FUNCTION_BLOCK Delta
VAR_INPUT
	MotionParameters	: DeltaMotionParameters_typ;			// Motion parameters used by internal motion function blocks	
	myMCSOverride: LREAL := 10.0;
	xSetOverride: BOOL;
	lrGrpOverride: MC_LREAL := 1.0;
	fbMC_GroupSetOverride : MC_GroupSetOverride;		
END_VAR

VAR_OUTPUT
	
	Ready				: BOOL;
	Busy				: BOOL;
	
	Error				: BOOL;
	ErrorID				: UDINT;
	ErrorOrigin			: STRING;	
		
	internalKinChanNCtoPLC	AT %I* : NCTOPLC_NCICHANNEL_REF;
	internalKinChanPLCtoNC	AT %Q* : PLCTONC_NCICHANNEL_REF;
		btest2: BOOL;	
	InKinematicsGroup		: BOOL;	
	InCoordinatedGroup		: BOOL;
	
	InSyncWithConveyor		: BOOL;

	//IdentInKinGroup			: UDINT;
	//IdentInCMGroup			: UDINT; 	
	
	ACS_A_REF	: AXIS_REF;
	ACS_B_REF	: AXIS_REF;
	ACS_C_REF	: AXIS_REF;
	
	MCS_X_REF	: AXIS_REF;
	MCS_Y_REF	: AXIS_REF;
	MCS_Z_REF	: AXIS_REF;
END_VAR
VAR
	
	{attribute 'instance-path'}
	{attribute 'no-init'}
	InstancePath			: STRING;
	btest: BOOL;
	AirVariable				AT %Q* : BOOL;
	
	internalEnable			: BOOL;
	internalDisable			: BOOL;
	
	//internalCurrentMoveType	: DeltaCommandType_enum;
	
	internalState			: DeltaState_enum;
	
	internalSetCoordTrafoDone	: BOOL;
	internalMovePathDone		: BOOL;

	
	internalInitObjPos		: ARRAY [1..3] OF MC_LREAL := [0,0,0];
	internalAxesList		: ST_KinAxes;
	internalCMGroup			: AXES_GROUP_REF;
	
	internalTrackAxis		: REFERENCE TO AXIS_REF;
	
	internalPathBuffer		: ARRAY[0..32767] OF BYTE;
	internalPathData		: MC_PATH_DATA_REF( ADR( internalPathBuffer ), SIZEOF( internalPathBuffer ));
		
	externalRoute			: REFERENCE TO Route;	

	internalActiveCoordRef	: MC_COORD_REF;		

	// Internal function blocks
	fbReset_MCS_X			: MC_Reset;
	fbReset_MCS_Y			: MC_Reset;
	fbReset_MCS_Z			: MC_Reset;
	
	fbReset_ACS_A			: MC_Reset;
	fbReset_ACS_B			: MC_Reset;
	fbReset_ACS_C			: MC_Reset;
	
	fbPower_MCS_X			: MC_Power;
	fbPower_MCS_Y			: MC_Power;
	fbPower_MCS_Z			: MC_Power;
	
	fbPower_ACS_A			: MC_Power;
	fbPower_ACS_B			: MC_Power;
	fbPower_ACS_C			: MC_Power;	
	
	fbAddAxisToGrp			: ARRAY[0..2] OF MC_AddAxisToGroup;
	fbGroupEnable			: MC_GroupEnable;
	
	fbKinConfigGroup		: FB_KinConfigGroup; 
	fbKinResetGroup			: FB_KinResetGroup;
	
	fbTrackBelt				: MC_TrackConveyorBelt;
	
	fbSetCoordTrafo			: MC_SetCoordinateTransform;
	fbMoveLinearPrep		: MC_MoveLinearAbsolutePreparation;
	fbMovePath				: MC_MovePath;
	fbMovePathExt			: MC_MovePath;
END_VAR

METHOD Cyclic : BOOL
VAR_IN_OUT
	//	KinematicGroup		: NCTOPLC;
END_VAR
VAR
	i: USINT;

END_VAR
CASE internalState OF
	DL_IDLE:	// ------------------------------------------------------- idle state
	
		Ready		:= FALSE;
		Busy		:= FALSE;
		
		internalDisable		:= FALSE;
		IF internalEnable THEN
			internalEnable		:= FALSE;
			internalState		:= DL_RESET;
		END_IF
	
	DL_RESET:	// ------------------------------------------------------- resets all axis objects
	
		Ready		:= FALSE;
		Busy		:= TRUE;
		Error		:= FALSE;
		ErrorID		:= 0;
		
		fbReset_MCS_X.Execute		:= TRUE;
		fbReset_MCS_Y.Execute		:= TRUE;
		fbReset_MCS_Z.Execute		:= TRUE;		
		
		fbReset_ACS_A.Execute		:= TRUE;
		fbReset_ACS_B.Execute		:= TRUE;
		fbReset_ACS_C.Execute		:= TRUE;
		
		IF fbReset_MCS_X.Done AND
			fbReset_MCS_Y.Done AND
			fbReset_MCS_Z.Done AND
			fbReset_ACS_A.Done AND
			fbReset_ACS_B.Done AND
			fbReset_ACS_C.Done THEN
			
			fbReset_MCS_X.Execute		:= FALSE;
			fbReset_MCS_Y.Execute		:= FALSE;
			fbReset_MCS_Z.Execute		:= FALSE;		
		
			fbReset_ACS_A.Execute		:= FALSE;
			fbReset_ACS_B.Execute		:= FALSE;
			fbReset_ACS_C.Execute		:= FALSE;
			
			internalState	:= DL_POWER_AXES;
			
		ELSIF fbReset_MCS_X.Error OR
			fbReset_MCS_Y.Error OR
			fbReset_MCS_Z.Error OR
			fbReset_ACS_A.Error OR
			fbReset_ACS_B.Error OR
			fbReset_ACS_C.Error THEN
			
			ErrorID; // TODO add whatever the error was for that block
			ErrorOrigin		:= CONCAT( InstancePath, '.fbReset' );
			internalState	:= DL_ERROR; 		
		END_IF
		
	DL_POWER_AXES:	// --------------------------------------------------- energizes all axis objects
	
		Ready		:= FALSE;
		Busy		:= TRUE;
		Error		:= FALSE;
		ErrorID		:= 0;

			fbPower_MCS_X.Enable	:= TRUE;
			fbPower_MCS_Y.Enable	:= TRUE;
			fbPower_MCS_Z.Enable	:= TRUE;
			
			fbPower_MCS_X.Enable_Positive	:= TRUE;
			fbPower_MCS_Y.Enable_Positive	:= TRUE;
			fbPower_MCS_Z.Enable_Positive	:= TRUE;
			
			fbPower_MCS_X.Enable_Negative	:= TRUE;
			fbPower_MCS_Y.Enable_Negative	:= TRUE;
			fbPower_MCS_Z.Enable_Negative	:= TRUE;
			
			fbPower_ACS_A.Enable	:= TRUE;
			fbPower_ACS_B.Enable	:= TRUE;
			fbPower_ACS_C.Enable	:= TRUE;
			
			fbPower_ACS_A.Enable_Positive	:= TRUE;
			fbPower_ACS_B.Enable_Positive	:= TRUE;
			fbPower_ACS_C.Enable_Positive	:= TRUE;
			
			fbPower_ACS_A.Enable_Negative	:= TRUE;
			fbPower_ACS_B.Enable_Negative	:= TRUE;
			fbPower_ACS_C.Enable_Negative	:= TRUE;
			
			fbPower_MCS_X.Override		:= myMCSOverride;
			fbPower_MCS_Y.Override		:= myMCSOverride;
			fbPower_MCS_Z.Override		:= myMCSOverride;
			
			IF fbPower_MCS_X.Status AND
				fbPower_MCS_Y.Status AND
				fbPower_MCS_Z.Status AND
				fbPower_ACS_A.Status AND
				fbPower_ACS_B.Status AND
				fbPower_ACS_C.Status THEN
				
				internalState	:= DL_SET_IK;
				
			ELSIF fbPower_MCS_X.Error OR
				fbPower_MCS_Y.Error OR
				fbPower_MCS_Z.Error OR
				fbPower_ACS_A.Error OR
				fbPower_ACS_B.Error OR
				fbPower_ACS_C.Error THEN
				
				ErrorID;	// TODO add whatever the error was that block
				ErrorOrigin		:= CONCAT( InstancePath, '.fbPower');
				internalState	:= DL_ERROR;
			END_IF

	
	DL_SET_IK:	// ------------------------------------------------------- enables the inverse kinematics transformation
	
		Ready		:= FALSE;
		Busy		:= TRUE;
		Error		:= FALSE;
		ErrorID		:= 0;

		internalAxesList.nAxisIdsAcs[1]		:= ACS_A_REF.NcToPlc.AxisId;
		internalAxesList.nAxisIdsAcs[2]		:= ACS_B_REF.NcToPlc.AxisId;
		internalAxesList.nAxisIdsAcs[3]		:= ACS_C_REF.NcToPlc.AxisId;
		
		internalAxesList.nAxisIdsMcs[1]		:= MCS_X_REF.NcToPlc.AxisId;
		internalAxesList.nAxisIdsMcs[2]		:= MCS_Y_REF.NcToPlc.AxisId;
		internalAxesList.nAxisIdsMcs[3]		:= MCS_Z_REF.NcToPlc.AxisId;
		
		fbKinConfigGroup.bExecute			:= TRUE;
		fbKinConfigGroup.bCartesianMode		:= TRUE;
	
	
		IF fbKinConfigGroup.bDone THEN
		//	fbKinConfigGroup.bExecute		:= FALSE;
			internalState					:= DL_DEBUG; //DL_ADD_AXES_TO_CM; // 
		ELSIF fbKinConfigGroup.bError THEN
			ErrorID			:= fbKinConfigGroup.nErrorId;
			ErrorOrigin		:= CONCAT(InstancePath,'.fbKinConfigGroup');
			internalState	:= DL_ERROR;
		END_IF;

		
	DL_ADD_AXES_TO_CM:	// ----------------------------------------------- adds MCS axes to CM Group
	
		Ready		:= FALSE;
		Busy		:= TRUE;
		Error		:= FALSE;
		ErrorID		:= 0;

			fbAddAxisToGrp[0].IdentInGroup	:= MCS_X;
			// fbAddAxisToGrp[0].Axis			:= MCS_X_REF;
			
			fbAddAxisToGrp[1].IdentInGroup	:= MCS_Y;
			// fbAddAxisToGrp[1].Axis			:= MCS_Y_REF;	
			
			fbAddAxisToGrp[2].IdentInGroup	:= MCS_Z;
			// fbAddAxisToGrp[2].Axis			:= MCS_Z_REF;
			
			FOR i := 0 TO 2 DO
				fbAddAxisToGrp[i].Execute		:= TRUE;
			END_FOR
			
			IF fbAddAxisToGrp[0].Done AND
				fbAddAxisToGrp[1].Done AND
				fbAddAxisToGrp[2].Done THEN
				
				fbAddAxisToGrp[0].Execute	:= FALSE;
				fbAddAxisToGrp[1].Execute	:= FALSE;
				fbAddAxisToGrp[2].Execute	:= FALSE;
				
				internalState	:= DL_ENABLE_CM;
				
			ELSIF fbAddAxisToGrp[0].Error OR
				fbAddAxisToGrp[1].Error OR
				fbAddAxisToGrp[2].Error THEN
				
				fbAddAxisToGrp[0].Execute	:= FALSE;
				fbAddAxisToGrp[1].Execute	:= FALSE;
				fbAddAxisToGrp[2].Execute	:= FALSE;
				
				ErrorID;		// todo : add whichever block errored
				ErrorOrigin		:= CONCAT(InstancePath,'.fbAddAxisToGrp');
				internalState	:= DL_ERROR;
			END_IF

	DL_ENABLE_CM:	// ------------------------------------------------------- enables the coordinated motion group
	
		Ready		:= FALSE;
		Busy		:= TRUE;
		Error		:= FALSE;
		ErrorID		:= 0;
		
			fbGroupEnable.Execute		:= TRUE;
			
			IF fbGroupEnable.Done THEN
				internalState	:= DL_RUN;
			ELSIF fbGroupEnable.Error THEN
				ErrorID			:= fbGroupEnable.ErrorId;
				ErrorOrigin		:= CONCAT(InstancePath,'.fbGroupEnable');
				internalState	:= DL_ERROR;
			END_IF
		
	DL_RUN:	// --------------------------------------------------------------- Delta running, ready for commands
	
		Ready		:= TRUE;
		Busy		:= FALSE;
		Error		:= FALSE;
		ErrorID		:= 0;
				
		// reset all commanded function blocks when the execute is recieved
		IF fbSetCoordTrafo.Busy OR fbSetCoordtrafo.CommandAborted THEN
			fbSetCoordTrafo.Execute		:= FALSE;
		ELSIF fbMovePath.Busy OR fbMovePath.CommandAborted THEN
			fbMovePath.Execute			:= FALSE;
		ELSIF fbMovePathEXT.Busy OR fbMovePathEXT.CommandAborted THEN
			fbMovePath.Execute			:= FALSE;
		ELSIF fbTrackBelt.Active OR fbTrackBelt.CommandAborted THEN
			fbTrackBelt.Execute			:= FALSE;
		END_IF
		
		// and catch all internal function block errors
		IF fbSetCoordTrafo.Error THEN
			ErrorID			:= fbSetCoordTrafo.ErrorId;
			ErrorOrigin		:= CONCAT( InstancePath, '.fbSetCoordTrafo' );
			internalState	:= DL_ERROR;
		ELSIF fbMovePath.Error THEN
			ErrorID			:= fbMovePath.ErrorId;
			ErrorOrigin		:= CONCAT( InstancePath, '.fbMovePath' );
			internalState	:= DL_ERROR;
		ELSIF fbMovePathEXT.Error THEN
			ErrorID			:= fbMovePathEXT.ErrorId;
			ErrorOrigin		:= CONCAT( InstancePath, '.fbMovePathEXT' );
			internalState	:= DL_ERROR;
		ELSIF fbTrackBelt.Error THEN
			ErrorID			:= fbMovePath.ErrorId;
			ErrorOrigin		:= CONCAT( InstancePath, '.fbMovePath' );
			internalState	:= DL_ERROR;
		END_IF
	
	DL_ERROR:	// ----------------------------------------------------------- Error state
	
		Ready		:= FALSE;
		Busy		:= FALSE;
		Error		:= TRUE;
	
END_CASE

fbReset_ACS_A( Axis := ACS_A_REF );
fbReset_ACS_B( Axis := ACS_B_REF );
fbReset_ACS_C( Axis := ACS_C_REF );
fbReset_MCS_X( Axis := MCS_X_REF );
fbReset_MCS_Y( Axis := MCS_Y_REF );
fbReset_MCS_Z( Axis := MCS_Z_REF );

fbPower_ACS_A( Axis := ACS_A_REF );
fbPower_ACS_B( Axis := ACS_B_REF );
fbPower_ACS_C( Axis := ACS_C_REF );
fbPower_MCS_X( Axis := MCS_X_REF );
fbPower_MCS_Y( Axis := MCS_Y_REF );
fbPower_MCS_Z( Axis := MCS_Z_REF );

fbAddAxisToGrp[0]( AxesGroup := internalCMGroup, Axis := MCS_X_REF );
fbAddAxisToGrp[1]( AxesGroup := internalCMGroup, Axis := MCS_Y_REF );
fbAddAxisToGrp[2]( AxesGroup := internalCMGroup, Axis := MCS_Z_REF );

fbGroupEnable( AxesGroup := internalCMGroup );

fbKinConfigGroup( stAxesList := internalAxesList, stKinRefIn := internalKinChanNCtoPLC );
fbKinResetGroup( stKinRefIn := internalKinChanNCtoPLC, stAxesList := internalAxesList );

fbSetCoordTrafo( AxesGroup := internalCMGroup );

fbMovePath( AxesGroup := internalCMGroup, PathData := internalPathData );
fbMovePathEXT( AxesGroup := internalCMGroup, PathData := externalRoute.PathData );

fbMC_GroupSetOverride(
	AxesGroup:= internalCMGroup, 
	Enable:= xSetOverride, 
	VelFactor:= lrGrpOverride, 
	Enabled=> , 
	Busy=> , 
	Error=> , 
	ErrorId=> , 
	ActualVelFactor=> );
END_METHOD

METHOD Disable : BOOL
VAR_INPUT
END_VAR
END_METHOD

METHOD DisableAir : BOOL
VAR_INPUT
END_VAR
AirVariable	:= FALSE;
END_METHOD

METHOD Enable : BOOL
VAR_INPUT
END_VAR
IF internalState = DL_IDLE THEN
	internalEnable		:= TRUE;
END_IF;
END_METHOD

METHOD EnableAir : BOOL
VAR_INPUT
END_VAR
AirVariable	:= TRUE;
END_METHOD

METHOD ExecuteRoute : BOOL
VAR_INPUT
	Route		: REFERENCE TO Route;
END_VAR
externalRoute			REF= Route;
fbMovePathEXT.Execute	:= TRUE;
END_METHOD

METHOD MoveDirectTo : BOOL
VAR_INPUT
	X			: LREAL;
	Y			: LREAL;
	Z			: LREAL;
END_VAR
VAR
	posVector			: ARRAY[0..2] OF LREAL;
	toleranceBall		: ARRAY[0..1] OF LREAL;
END_VAR
// clear any existing waypoints in the path buffer
internalPathData.ClearPath();

// add a single point at the destination
posVector[0]	:= X;
posVector[1]	:= Y;
posVector[2]	:= Z;

// blending radii follows a ratio recommendation from infosys
toleranceBall[0]	:= 0.5 * MotionParameters.BlendingRadius;
toleranceBall[1]	:= MotionParameters.BlendingRadius;

fbMoveLinearPrep.Position			:= ADR( posVector );
fbMoveLinearPrep.PositionCount		:= 3;
fbMoveLinearPrep.Velocity			:= MotionParameters.Velocity;
fbMoveLinearPrep.Acceleration		:= MotionParameters.Acceleration;
fbMoveLinearPrep.Deceleration		:= MotionParameters.Deceleration;
fbMoveLinearPrep.Jerk				:= MotionParameters.Jerk;
fbMoveLinearPrep.BufferMode			:= mcBlendingPrevious;

fbMoveLinearPrep.TransitionMode				:= mcTransModeCornerDistanceAdvanced;
fbMoveLinearPrep.TransitionParameter		:= ADR( toleranceBall );
fbMoveLinearPrep.TransitionParameterCount	:= 2;
fbMoveLinearPrep.InvokeId					:= 100;

fbMoveLinearPrep( PathData := internalPathData );

// execute mc_movepath
fbMovePath.Execute	:= TRUE;

fbMovePath( AxesGroup := internalCMGroup, PathData := internalPathData );
END_METHOD

PROPERTY MovePathDone : BOOL
GET
MovePathDone		:= fbMovePath.Done;
END_GET
END_PROPERTY

METHOD Reset : BOOL
VAR_INPUT
END_VAR
internalState := DL_IDLE;
END_METHOD

METHOD ReturnHome : BOOL
VAR_INPUT
END_VAR
// Zero is home, right?
THIS^.MoveDirectTo( 0, 100, 50);
END_METHOD

METHOD SetAcceleration : BOOL
VAR_INPUT
	Acceleration	: LREAL;
END_VAR
// prevents a negative value from being accepted
MotionParameters.Acceleration		:= LIMIT( 0, Acceleration, 1E300 );
END_METHOD

METHOD SetCoordTrafo : BOOL
VAR_INPUT
	CoordRef	: MC_COORD_REF;
END_VAR
// Set the function block to change coordinate reference frame
fbSetCoordTrafo.Execute				:= TRUE;
fbSetCoordTrafo.CoordTransform		:= CoordRef;	

internalActiveCoordRef				:= CoordRef;

fbSetCoordTrafo( AxesGroup := internalCMGroup );
END_METHOD

PROPERTY SetCoordTrafoDone : BOOL
GET
SetCoordTrafoDone	:= fbSetCoordTrafo.Done;
END_GET
END_PROPERTY

METHOD SetDeceleration : BOOL
VAR_INPUT
	Deceleration		: LREAL;
END_VAR

// prevent a negative value from being accepted
MotionParameters.Deceleration	:= LIMIT( 0, Deceleration, 1E300 );
END_METHOD

METHOD SetJerk : BOOL
VAR_INPUT
	Jerk		: LREAL;
END_VAR

// Prevents a negative value from being accepted.
MotionParameters.Jerk		:= LIMIT( 0, Jerk, 1E300 );
END_METHOD

METHOD SetVelocity : BOOL
VAR_INPUT
	Velocity		: LREAL;
END_VAR

// Prevents a negative value from being accepted
MotionParameters.Velocity		:= LIMIT( 0, Velocity, 1E300 );
END_METHOD

METHOD TrackConveyor : BOOL
VAR_INPUT
	MasterRefPos		: MC_LREAL;
	TrackAxis			: REFERENCE TO AXIS_REF;
	CoordFrame			: MC_COORD_REF;
END_VAR


internalTrackAxis		REF= TrackAxis;

//initialObjectPos[1]		:= 0;
//initialObjectPos[2]		:= 0;
//initialObjectPos[3]		:= 0;

fbTrackBelt.CoordTransform			:= CoordFrame;
fbTrackBelt.InitialObjectPos		:= ADR( internalInitObjPos );
fbTrackBelt.InitialObjectPosCount	:= 3;
fbTrackBelt.MasterRefPos			:= MasterRefPos;

fbTrackBelt.Velocity		:= MotionParameters.Velocity;
fbTrackBelt.Acceleration	:= MotionParameters.Acceleration;
fbTrackBelt.Deceleration	:= MotionParameters.Deceleration;
fbTrackBelt.Jerk			:= MotionParameters.Jerk;

fbTrackBelt.Execute		:= TRUE;

fbTrackBelt( AxesGroup := internalCMGroup, ConveyorBelt := internalTrackAxis );
END_METHOD

PROPERTY TrackConveyorActive : BOOL
GET
TrackConveyorActive		:= fbTrackBelt.InSync;
END_GET
END_PROPERTY

METHOD TraverseAtHeightTo : BOOL
VAR_INPUT
	X			: LREAL;
	Y			: LREAL;
	Z			: LREAL;
	TraverseZ	: LREAL;
END_VAR
VAR
	posVector		: ARRAY[0..2] OF LREAL;
	toleranceBall	: ARRAY[0..1] OF LREAL;
END_VAR
// clear any existing waypoints in the path buffer
internalPathData.ClearPath();

toleranceBall[0]	:= 0.5 * MotionParameters.BlendingRadius;
toleranceBall[1]	:= MotionParameters.BlendingRadius;

fbMoveLinearPrep.PositionCount		:= 3;
fbMoveLinearPrep.Velocity			:= MotionParameters.Velocity;
fbMoveLinearPrep.Acceleration		:= MotionParameters.Acceleration;
fbMoveLinearPrep.Deceleration		:= MotionParameters.Deceleration;
fbMoveLinearPrep.Jerk				:= MotionParameters.Jerk;
fbMoveLinearPrep.BufferMode			:= mcBlendingPrevious;

fbMoveLinearPrep.TransitionMode				:= mcTransModeCornerDistanceAdvanced;
fbMoveLinearPrep.TransitionParameter		:= ADR( toleranceBall );
fbMoveLinearPrep.TransitionParameterCount	:= 2;
fbMoveLinearPrep.InvokeId					:= 100;

// add a vertical movement to the traverse height
posVector[0]		:= MCS_X_REF.NcToPlc.ActPos; 
posVector[1]		:= MCS_Y_REF.NcToPlc.ActPos;
posVector[2]		:= TraverseZ;

fbMoveLinearPrep.Position		:= ADR( posVector );
fbMoveLinearPrep( PathData := internalPathData );

// add a traversal move to a point above/below the destination
posVector[0]		:= X;	// destination X
posVector[1]		:= Y;	// destination Y
posVector[2]		:= TraverseZ;	// traversal height

fbMoveLinearPrep.Position		:= ADR( posVector );
fbMoveLinearPrep( PathData := internalPathData );

// add a vertical move to the destination itself
posVector[0]		:= X;
posVector[1]		:= Y;
posVector[2]		:= Z;

fbMoveLinearPrep.Position		:= ADR( posVector );
fbMoveLinearPrep( PathData := internalPathData );

// execute mc_movepath
fbMovePath.Execute	:= TRUE;

// Call once for Busy output
fbMovePath( AxesGroup := internalCMGroup, PathData := internalPathData );
END_METHOD

END_FUNCTION_BLOCK

(* stored: Version 1.1.0.1, ProductVersion 3.1.4024.11
   POU Delta: Id {492a738f-fc6d-4715-b733-4ea1b08e2312}, SpecialFunc None
   Folder Methods: Id {a2d46a1e-7a9e-44a1-9a9c-487d94df0d8d}
   Folder Properties: Id {68d119c4-1e71-4d9e-a63e-63c332a25cde}
   Method Cyclic: Id {08a56dcb-206a-41ec-ac0a-83b543ba62a8}
   Method Disable: Id {f8852278-a902-41fb-8b1a-a53ea61cbd64}
   Method DisableAir: Id {74258680-12ce-4520-8174-1e7920fb856e}
   Method Enable: Id {f4887e95-9084-4d7c-8994-4709154d6c02}
   Method EnableAir: Id {64a72ef1-4b6d-4e9c-8d63-cad412c5e0f0}
   Method ExecuteRoute: Id {0f1c4d90-fa0e-4ee0-9899-a01e330415e2}
   Method MoveDirectTo: Id {610f0aa4-e8d8-4a0e-b42c-d66003cd2595}
   Property MovePathDone: Id {dd8dbeba-3161-4047-8127-ea64b21675c1}
   Get Get: Id {7df17e80-557a-41df-8651-9ebd7ef9a364}
   Method Reset: Id {53b97b6c-d929-489a-b91b-ad9f50847a2c}
   Method ReturnHome: Id {4a762706-93bb-4e83-8b35-d2c1fae7dbb3}
   Method SetAcceleration: Id {92321fb0-df12-41a8-a2c8-436a5c15bd2a}
   Method SetCoordTrafo: Id {6bf0c707-36e2-400d-ba6a-1409a4ef623e}
   Property SetCoordTrafoDone: Id {71fa1ee3-447a-48eb-933c-e282e4815b89}
   Get Get: Id {dca464b8-bfd9-4ed6-aeb3-8b7143978587}
   Method SetDeceleration: Id {45bf2e83-ee20-441b-9e55-4922a9803644}
   Method SetJerk: Id {4ef692c6-1a95-42ab-8a1b-79d9a2e89408}
   Method SetVelocity: Id {24facd4e-7d50-487f-9c83-08886c6f20a6}
   Method TrackConveyor: Id {2816da83-ed23-43ce-a0b7-378371c4fed3}
   Property TrackConveyorActive: Id {f310fd5c-ce55-4c44-b116-740d45e473da}
   Get Get: Id {6306f1a7-01b5-47a4-929e-037481165b52}
   Method TraverseAtHeightTo: Id {09ea2bd6-1601-4fea-823b-7e058bcdd11a} *)
